// TIA Portal project "TIA Portal Project" (V20)

(* hardware
DEVICE "S7-1500/ET200MP station_1"  S7-1500 station
   slot 0: "Rail_0"  Rack  6ES7 590-1***0-0AA0
   slot 1: "PLC_1"  CPU 1515-2 PN  6ES7 515-2AN03-0AB0  V4.0
      slot 3: "CPU display_1"  6ES7591-1BA00-0AA0
      slot 32768: "PROFINET interface_1"  X1
         slot 32769: "Port_1"  X1 P1
         slot 32770: "Port_2"  X1 P2
      slot 33024: "PROFINET interface_2"  X2
         slot 33025: "Port_1"  X2 P1
      slot 34817: "Virtual CP interface port_1"  Virtual CP interface port  Virtual CP interface port FW V4.0
   slot 2: "DI 16x24VDC BA_1"  DI 16x24VDC BA  6ES7 521-1BH10-0AA0  V1.1
   slot 3: "DQ 16x24VDC/0.5A BA_1"  DQ 16x24VDC/0.5A BA  6ES7 522-1BH10-0AA0  V1.1
   slot 4: "AI 8xU/I HS_1"  AI 8xU/I HS  6ES7 531-7NF10-0AB0  V2.1
   slot 5: "AQ 8xU/I HS_1"  AQ 8xU/I HS  6ES7 532-5HF00-0AB0  V2.2
*)

// ===== PLC "PLC_1"  CPU 1515-2 PN =====

VAR_GLOBAL   // PLC tag table "Default tag table"
   "Start" AT %I0.0 : Bool;
   "Stop" AT %I0.1 : Bool;
   "Program_On" AT %Q0.1 : Bool;
   "AutoON" AT %M100.0 : Bool;   // AutoON
END_VAR

FUNCTION "Program" : Void   // FC1, LAD
{ S7_Optimized_Access := 'TRUE' }
VERSION : 0.1
BEGIN

REGION Network 1
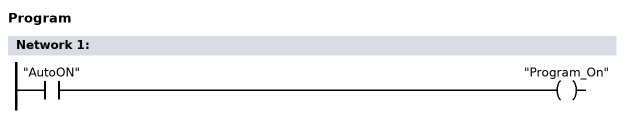
   RUNG wire#powerrail
      Contact( "AutoON" )
      Coil( "Program_On" )
   END_RUNG
   // the same network as SCL:
   "Program_On" := "AutoON";
END_REGION
END_FUNCTION

FUNCTION "F_Safety" : Void   // FC2, LAD
{ S7_Optimized_Access := 'TRUE' }
VERSION : 0.1
BEGIN

REGION Network 1
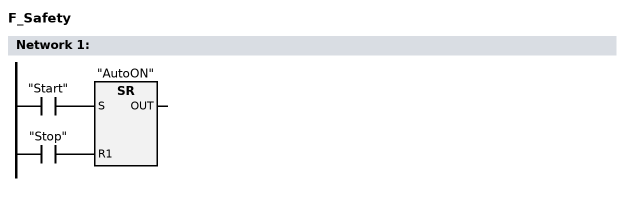
   RUNG wire#powerrail
      Contact( "Start" )
      S_SR(operand := "AutoON", r1 := wire#w1)
   END_RUNG
   RUNG wire#powerrail
      Contact( "Stop" )
   END_RUNG wire#w1
   // the same network as SCL:
   IF "Start" THEN
       "AutoON" := TRUE;   // SR flip-flop
   END_IF;
   IF "Stop" THEN "AutoON" := FALSE; END_IF;
END_REGION
END_FUNCTION

ORGANIZATION_BLOCK "Main"   // OB1, LAD, ProgramCycle
TITLE = "Main Program Sweep (Cycle)"
{ S7_Optimized_Access := 'TRUE' }
VERSION : 0.1
   VAR_INPUT
      Initial_Call : Bool;   // Initial call of this OB
      Remanence : Bool;   // =True, if remanent data are available
   END_VAR
BEGIN
END_ORGANIZATION_BLOCK